TYPE DUT_HMI_EV_Diagnostic :
STRUCT
	Enable	 : BOOL;
	dFwdTime : UINT;
	dBwdTime : UINT;
	eStatus  : eEV_Status;
	Error 	 : BOOL;	
END_STRUCT
END_TYPE

(* stored: Version 1.1.0.1, ProductVersion 3.1.4024.13
   DUT DUT_HMI_EV_Diagnostic: Id {bef335ad-ddc5-43cd-8176-e7db73f79956} *)
